INTERFACE I_Mover

METHOD CycleUpdate : BOOL
VAR_INPUT
END_VAR
END_METHOD

PROPERTY distToEndOfTrack : Lreal
GET
END_GET
END_PROPERTY

METHOD Init : BOOL
VAR_INPUT
	XtsMover:  I_XtsXlMover1;
	XtsProcessingUnit :  I_XtsProcessingUnit1;

	
END_VAR
END_METHOD

METHOD JoinNearestTrack : BOOL

VAR_INPUT 
	aMcTracks : ARRAY[*] OF MC_PlanarTrack;
	Trackcount : UINT;
END_VAR
END_METHOD

METHOD LeaveSystemAt : BOOL
VAR_INPUT
	ConnectionOut: REFERENCE TO MC_PlanarTrackConnectionOut;	
	gap : LREAL; 		
END_VAR
END_METHOD

METHOD MoveOnTrack : BOOL
VAR_INPUT
	track: REFERENCE TO MC_PlanarTrack;	
	targetPos: LREAL;
	gap : LREAL; 

END_VAR
END_METHOD

PROPERTY MoverStopped : BOOL
GET
END_GET
SET
END_SET
END_PROPERTY

PROPERTY P_Dynamics : REFERENCE TO DynamicConstraint_PathXY;
GET
END_GET
END_PROPERTY

PROPERTY P_IsInitialized : bool
GET
END_GET
END_PROPERTY

PROPERTY P_MoverOTCID : OTCID
GET
END_GET
SET
END_SET
END_PROPERTY

PROPERTY P_PlanarFeedback : REFERENCE TO MC_PlanarFeedback
GET
END_GET
END_PROPERTY

PROPERTY P_PlanarMover :   REFERENCE TO  MC_PlanarMover
GET
END_GET
END_PROPERTY

PROPERTY P_SyncFeedback :  REFERENCE TO MC_PlanarFeedbackGearInPosOnTrackWithMasterMover
GET
END_GET
END_PROPERTY

PROPERTY P_TargetTrack : UDINT
GET
END_GET
SET
END_SET
END_PROPERTY

PROPERTY Rework : BOOL
GET
END_GET
SET
END_SET
END_PROPERTY

METHOD SyncToOtherMover : Bool
VAR_INPUT
	masterSyncPos : LREAL; // Position on the master track
	followerSyncPos : LREAL; // position on the follower track
	PlanarMoverToFollow: REFERENCE TO Tc3_Mc3PlanarMotion.MC_PlanarMover;
	masterTrack : REFERENCE TO Tc3_Mc3PlanarMotion.MC_PlanarTrack; 
	followerTrack : REFERENCE TO Tc3_Mc3PlanarMotion.MC_PlanarTrack; 
	velo :  REFERENCE TO LREAL; 
END_VAR
END_METHOD

METHOD  UpdateXtsTrack
VAR_INPUT
END_VAR
VAR

END_VAR
END_METHOD

PROPERTY XlProcessingUnit : I_XtsProcessingUnit1
GET
END_GET
END_PROPERTY

PROPERTY XtsComFeed : REFERENCE TO  XtsCommandFeedback
GET
END_GET
END_PROPERTY

PROPERTY XtsXlMover :  I_XtsXlMover1
GET
END_GET
END_PROPERTY

END_INTERFACE

(* stored: Version 1.1.0.1
   Itf I_Mover: Id {b268cb59-d99c-43ca-ba0f-41461eab83e4}
   Method CycleUpdate: Id {48e7b414-8a52-4904-8a2c-941ff8cf97f0}
   Property distToEndOfTrack: Id {54946fd7-00e4-4584-be84-948ea3635443}
   Get Get: Id {72f5bf45-38a7-4db3-85a2-cd77e7e3e0e0}
   Method Init: Id {70e27be2-2f8a-4a12-af9c-c87e7a1f6409}
   Method JoinNearestTrack: Id {1af77ee2-ffb0-46d3-b285-380f37f7d28e}
   Method LeaveSystemAt: Id {b24f1fa5-5146-4fc9-b97d-6c3d7849e67f}
   Method MoveOnTrack: Id {c4ca36ea-3628-4f8d-9779-76967292fe61}
   Property MoverStopped: Id {9803e80b-12ab-4e37-a4f8-315195184be1}
   Get Get: Id {2a3332aa-8658-4fa3-9f30-0f6bc046db6e}
   Set Set: Id {09465482-72a9-4047-a401-b7303e1e4a34}
   Property P_Dynamics: Id {a2d4066c-df4e-4534-b63b-1bcfe3693364}
   Get Get: Id {45b7255c-36dc-485f-87f9-8e7eaabd396d}
   Property P_IsInitialized: Id {809c04b6-b7db-4fb8-a7e6-29c53b002db8}
   Get Get: Id {a718d62b-bba8-464d-90ba-0ec43e78fd5e}
   Property P_MoverOTCID: Id {48d62f0a-81b1-4685-945a-1fd17f9606ba}
   Get Get: Id {f99e891b-2de5-41fe-8b1c-f0905de95a9f}
   Set Set: Id {f8a2dcde-e0e0-405c-9385-45717b5e9410}
   Property P_PlanarFeedback: Id {9e77b007-b995-4d4e-847f-52481bc8b65f}
   Get Get: Id {081f5294-b87e-4178-b95d-4508c49af3d5}
   Property P_PlanarMover: Id {fa6a8c9a-a607-48a6-a503-b7396c44d435}
   Get Get: Id {612fed8f-dbe1-4fd7-b02f-fa8abf96bee3}
   Property P_SyncFeedback: Id {44e12130-9d7b-42f1-8fbe-83c3e8bf9e21}
   Get Get: Id {d4c33880-d06d-4748-93ef-961feda12b5d}
   Property P_TargetTrack: Id {efe12142-6a27-4117-844c-b25d6699356f}
   Get Get: Id {c97343a2-cb69-4cb8-a50f-8b0d0fc63da3}
   Set Set: Id {eb872bda-1329-4f18-b45c-06f3807c5ce6}
   Property Rework: Id {0cbdc2c5-5567-4b77-b67c-5f6aa39ca7ad}
   Get Get: Id {3e2576da-ff58-4bce-81c6-db8a01090e8e}
   Set Set: Id {8ba65916-e99e-4e0b-8c93-c9e4c19a7a79}
   Method SyncToOtherMover: Id {53951dae-e642-4c0f-afd2-22812dd067a9}
   Method UpdateXtsTrack: Id {f15d0a33-41f6-42cf-a0d1-8e20b2064dca}
   Property XlProcessingUnit: Id {4fb3d0ec-89c3-4528-ba23-e01b215f5acc}
   Get Get: Id {37f03f3c-5775-4b0c-a635-c2033ace3510}
   Property XtsComFeed: Id {9b70f023-8c1f-45c7-92b4-2da0d8c5dc09}
   Get Get: Id {d2b3a28a-6116-4e27-ae7b-52ce23eb12f2}
   Property XtsXlMover: Id {bb8d0ca5-767e-4004-9c86-a2c6dc44ab36}
   Get Get: Id {23a9625f-4b2a-46c1-941c-9a84dc34c137} *)
